FUNCTION FLOOR (* This is a rounding function which returns the biggest possible integer which is less or equal to X. *)
  (* Standard: 61499-1 *)
  (* Version 1.0, 2026-09-17, Franz Höpfinger, Portiert aus OSCAT_basic FLOOR.TcPOU - Bereichspruefung (X >= 32767.0 / X <= -32768.0) schuetzt vor INT-Ueberlauf. *)
  PACKAGE OSCAT::Basic::POUs::Mathematical;
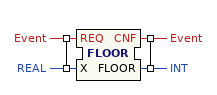
  EVENT_INPUT
    REQ WITH X;
  END_EVENT
  EVENT_OUTPUT
    CNF WITH FLOOR;
  END_EVENT
  VAR_INPUT
    X : REAL;
  END_VAR
  VAR_OUTPUT
    FLOOR : INT;
  END_VAR
  BODY IN ST:
PACKAGE OSCAT::Basic::POUs::Mathematical;

(* This is a rounding function which returns the biggest possible integer which is less or equal to X (clamped to INT range -32768..32767). *)
FUNCTION FLOOR : INT
VAR_INPUT
	X : REAL;
END_VAR

(*
 * version 1.1	21. mar. 2008 programmer 	hugo tested by		tobias
 * *
 * This is a rounding function which returns the biggest possible integer which is less or equal to X.
 * floor(3.14) = 3 floor(-3.14) = -4
 * Portiert 2026-09-17: Bereichspruefung schuetzt vor INT-Ueberlauf.
 *)
IF X >= 32767.0 THEN
	FLOOR := 32767;
ELSIF X <= -32768.0 THEN
	FLOOR := -32768;
ELSE
	FLOOR := REAL_TO_INT(X);
	IF FLOOR > X THEN
		FLOOR := FLOOR - 1;
	END_IF;
END_IF;

END_FUNCTION

(*
 * version 1.1	21. mar. 2008 programmer 	hugo tested by		tobias
 * *
 * This is a rounding function which returns the biggest possible integer which is less or equal to
 * X.
 * floor(3.14) = 3 floor(-3.14) = -4
 *)
  END_BODY
END_FUNCTION
